% RSLogix 500 project MDM UPGRADE - onsite 5-11-08.RSS, saved by version 7.00.00.19 %
PROJECT "UNTITLED"    % processor: MicroLogix 1200 %

PROGRAM FILES
  LAD 2 "MAIN"  10 rungs
  LAD 3 "SEQUENCE"  61 rungs
  LAD 4 "OUTPUTS"  12 rungs

DATA FILES
  O0 OUTPUT  4 elements
  I1 INPUT  4 elements
  S2 STATUS  66 elements
  B3 BINARY  4 elements
  T4 TIMER  3 elements
  C5 COUNTER  1 elements
  R6 CONTROL  1 elements
  N7 INTEGER  7 elements
  F8 FLOAT  1 elements
  N9 SEQ TIMES  100 elements

LADDER 2 "MAIN"
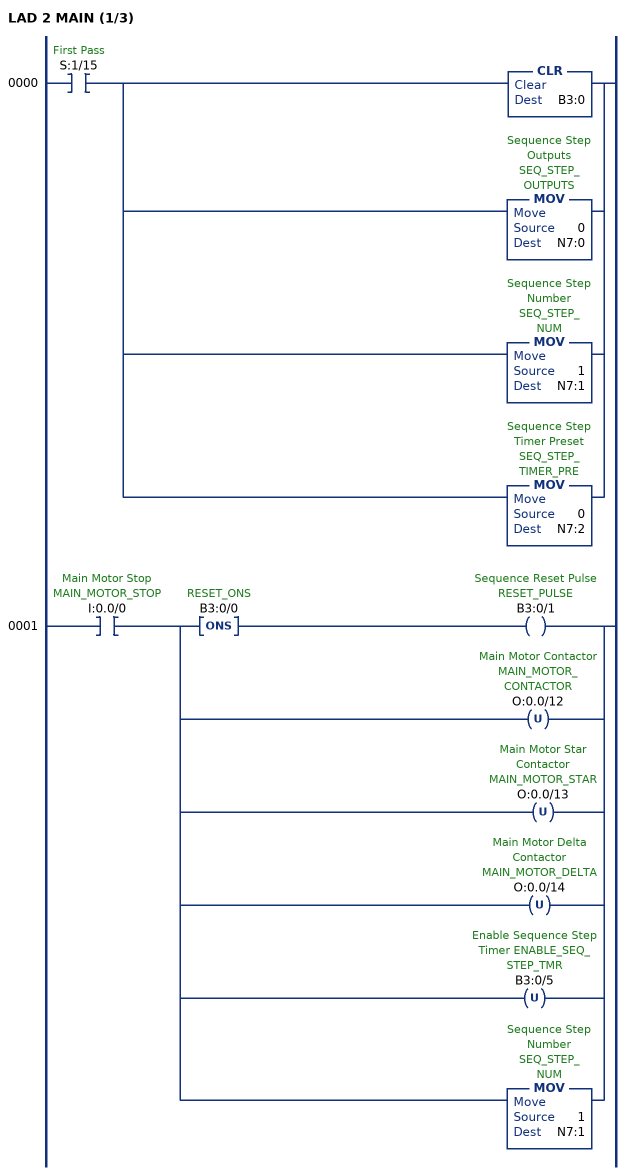
% Rung: 0 %
SOR XIC S:1/15 BST CLR B3:0 NXB MOV 0 N7:0 NXB MOV 1 N7:1 NXB MOV 0 N7:2 BND EOR
%   S:1/15  "First Pass" %
%   N7:0  SEQ_STEP_OUTPUTS  "Sequence Step Outputs" %
%   N7:1  SEQ_STEP_NUM  "Sequence Step Number" %
%   N7:2  SEQ_STEP_TIMER_PRE  "Sequence Step Timer Preset" %
% Rung: 1 %
SOR XIC I:0.0/0 BST ONS B3:0/0 OTE B3:0/1 NXB OTU O:0.0/12 NXB OTU O:0.0/13 NXB OTU O:0.0/14 NXB OTU B3:0/5 NXB MOV 1 N7:1 BND EOR
%   I:0.0/0  MAIN_MOTOR_STOP  "Main Motor Stop" %
%   B3:0/0  RESET_ONS %
%   B3:0/1  RESET_PULSE  "Sequence Reset Pulse" %
%   O:0.0/12  MAIN_MOTOR_CONTACTOR  "Main Motor Contactor" %
%   O:0.0/13  MAIN_MOTOR_STAR  "Main Motor Star Contactor" %
%   O:0.0/14  MAIN_MOTOR_DELTA  "Main Motor Delta Contactor" %
%   B3:0/5  ENABLE_SEQ_STEP_TMR  "Enable Sequence Step Timer" %
%   N7:1  SEQ_STEP_NUM  "Sequence Step Number" %

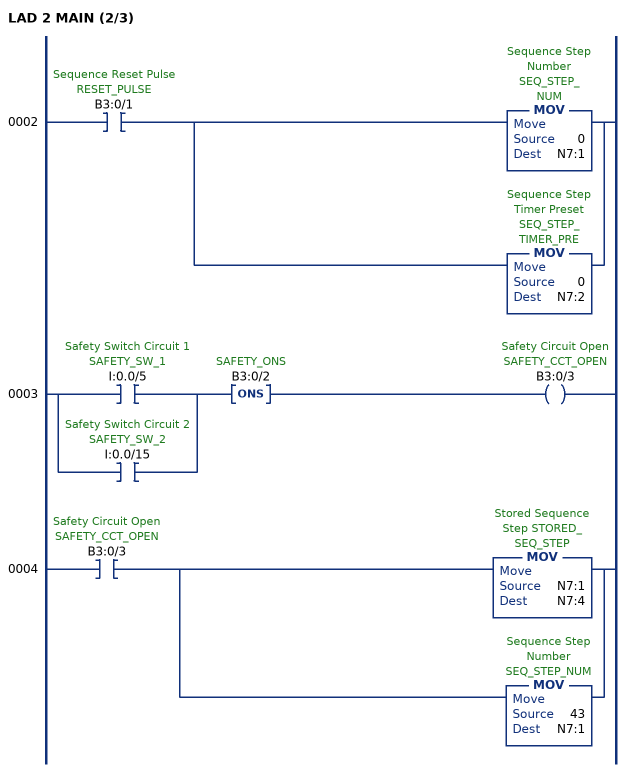
% Rung: 2 %
SOR XIC B3:0/1 BST MOV 0 N7:1 NXB MOV 0 N7:2 BND EOR
%   B3:0/1  RESET_PULSE  "Sequence Reset Pulse" %
%   N7:1  SEQ_STEP_NUM  "Sequence Step Number" %
%   N7:2  SEQ_STEP_TIMER_PRE  "Sequence Step Timer Preset" %
% Rung: 3 %
SOR BST XIC I:0.0/5 NXB XIC I:0.0/15 BND ONS B3:0/2 OTE B3:0/3 EOR
%   I:0.0/5  SAFETY_SW_1  "Safety Switch Circuit 1" %
%   I:0.0/15  SAFETY_SW_2  "Safety Switch Circuit 2" %
%   B3:0/2  SAFETY_ONS %
%   B3:0/3  SAFETY_CCT_OPEN  "Safety Circuit Open" %
% Rung: 4 %
SOR XIC B3:0/3 BST MOV N7:1 N7:4 NXB MOV 43 N7:1 BND EOR
%   B3:0/3  SAFETY_CCT_OPEN  "Safety Circuit Open" %
%   N7:1  SEQ_STEP_NUM  "Sequence Step Number" %
%   N7:4  STORED_SEQ_STEP  "Stored Sequence Step" %

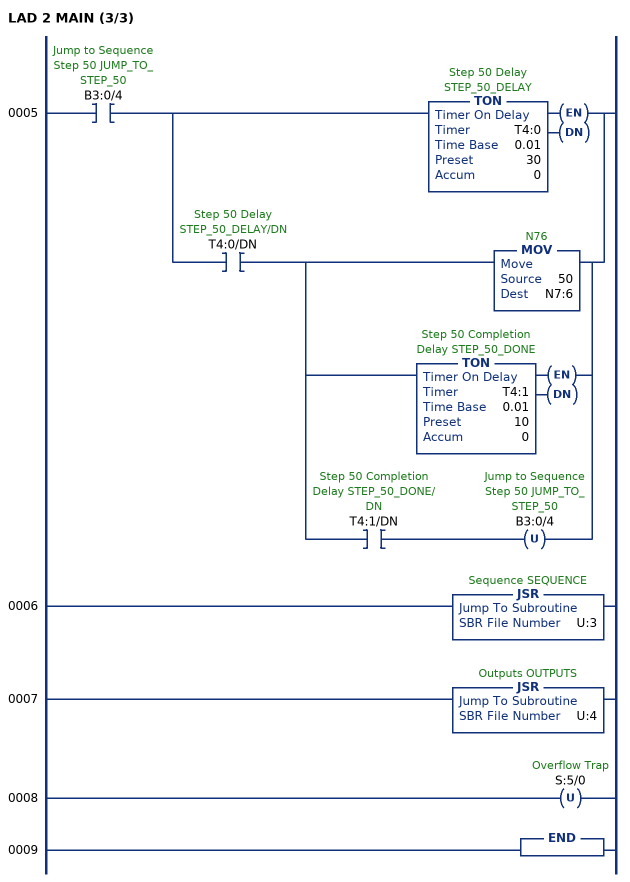
% Rung: 5 %
SOR XIC B3:0/4 BST TON T4:0 0.01 30 0 NXB XIC T4:0/DN BST MOV 50 N7:6 NXB TON T4:1 0.01 10 0 NXB XIC T4:1/DN OTU B3:0/4 BND BND EOR
%   B3:0/4  JUMP_TO_STEP_50  "Jump to Sequence Step 50" %
%   T4:0  STEP_50_DELAY  "Step 50 Delay" %
%   N7:6  N76 %
%   T4:1  STEP_50_DONE  "Step 50 Completion Delay" %
% Rung: 6 %
SOR JSR U:3 EOR
%   U:3  SEQUENCE  "Sequence" %
% Rung: 7 %
SOR JSR U:4 EOR
%   U:4  OUTPUTS  "Outputs" %
% Rung: 8 %
SOR OTU S:5/0 EOR
%   S:5/0  "Overflow Trap" %
% Rung: 9 %
SOR END EOR

LADDER 3 "SEQUENCE"
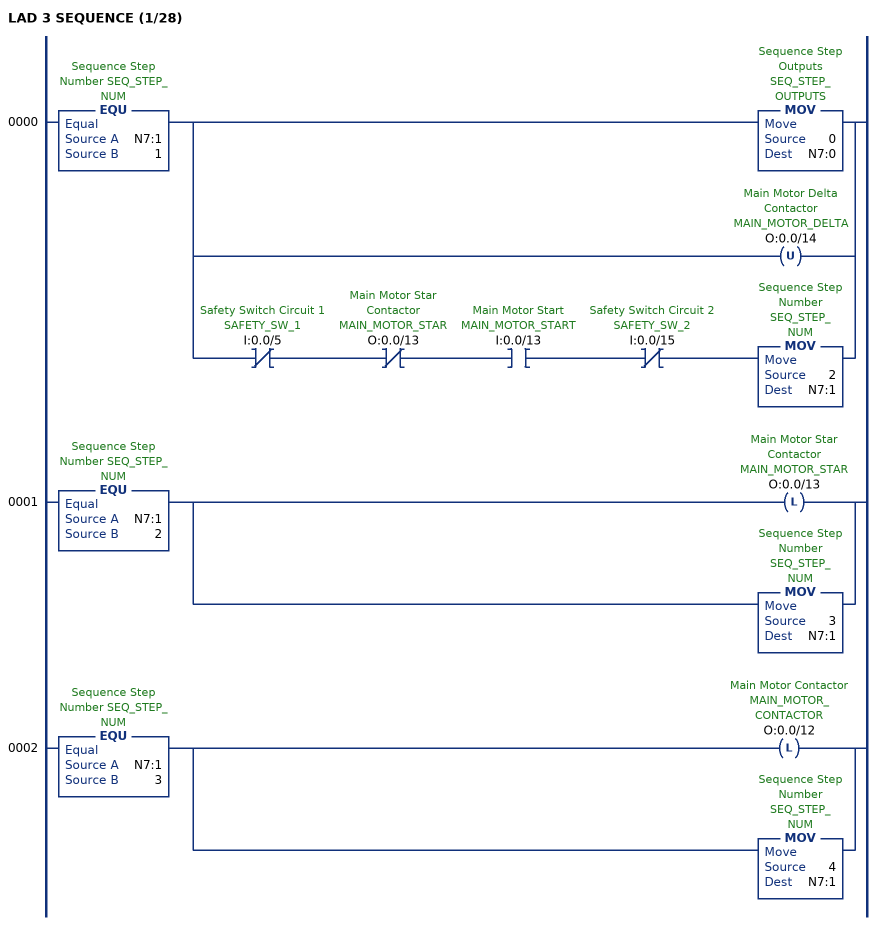
% Rung: 0 %
SOR EQU N7:1 1 BST MOV 0 N7:0 NXB OTU O:0.0/14 NXB XIO I:0.0/5 XIO O:0.0/13 XIC I:0.0/13 XIO I:0.0/15 MOV 2 N7:1 BND EOR
%   N7:1  SEQ_STEP_NUM  "Sequence Step Number" %
%   N7:0  SEQ_STEP_OUTPUTS  "Sequence Step Outputs" %
%   O:0.0/14  MAIN_MOTOR_DELTA  "Main Motor Delta Contactor" %
%   I:0.0/5  SAFETY_SW_1  "Safety Switch Circuit 1" %
%   O:0.0/13  MAIN_MOTOR_STAR  "Main Motor Star Contactor" %
%   I:0.0/13  MAIN_MOTOR_START  "Main Motor Start" %
%   I:0.0/15  SAFETY_SW_2  "Safety Switch Circuit 2" %
% Rung: 1 %
SOR EQU N7:1 2 BST OTL O:0.0/13 NXB MOV 3 N7:1 BND EOR
%   N7:1  SEQ_STEP_NUM  "Sequence Step Number" %
%   O:0.0/13  MAIN_MOTOR_STAR  "Main Motor Star Contactor" %
% Rung: 2 %
SOR EQU N7:1 3 BST OTL O:0.0/12 NXB MOV 4 N7:1 BND EOR
%   N7:1  SEQ_STEP_NUM  "Sequence Step Number" %
%   O:0.0/12  MAIN_MOTOR_CONTACTOR  "Main Motor Contactor" %

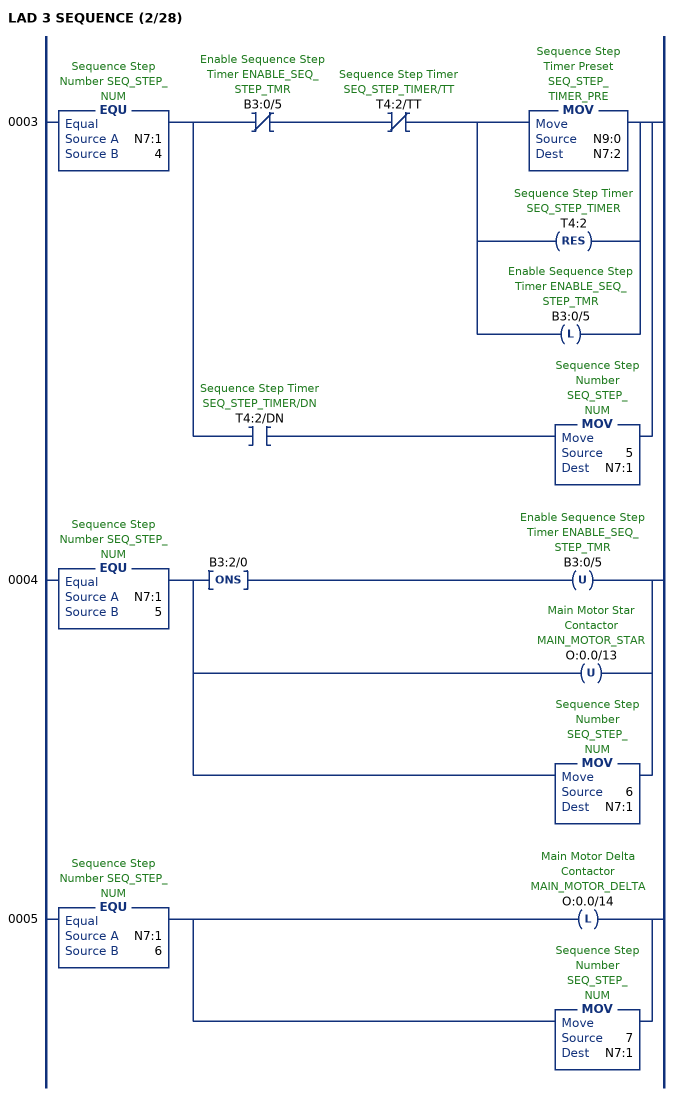
% Rung: 3 %
SOR EQU N7:1 4 BST XIO B3:0/5 XIO T4:2/TT BST MOV N9:0 N7:2 NXB RES T4:2 NXB OTL B3:0/5 BND NXB XIC T4:2/DN MOV 5 N7:1 BND EOR
%   N7:1  SEQ_STEP_NUM  "Sequence Step Number" %
%   B3:0/5  ENABLE_SEQ_STEP_TMR  "Enable Sequence Step Timer" %
%   T4:2  SEQ_STEP_TIMER  "Sequence Step Timer" %
%   N7:2  SEQ_STEP_TIMER_PRE  "Sequence Step Timer Preset" %
% Rung: 4 %
SOR EQU N7:1 5 BST ONS B3:2/0 OTU B3:0/5 NXB OTU O:0.0/13 NXB MOV 6 N7:1 BND EOR
%   N7:1  SEQ_STEP_NUM  "Sequence Step Number" %
%   B3:0/5  ENABLE_SEQ_STEP_TMR  "Enable Sequence Step Timer" %
%   O:0.0/13  MAIN_MOTOR_STAR  "Main Motor Star Contactor" %
% Rung: 5 %
SOR EQU N7:1 6 BST OTL O:0.0/14 NXB MOV 7 N7:1 BND EOR
%   N7:1  SEQ_STEP_NUM  "Sequence Step Number" %
%   O:0.0/14  MAIN_MOTOR_DELTA  "Main Motor Delta Contactor" %

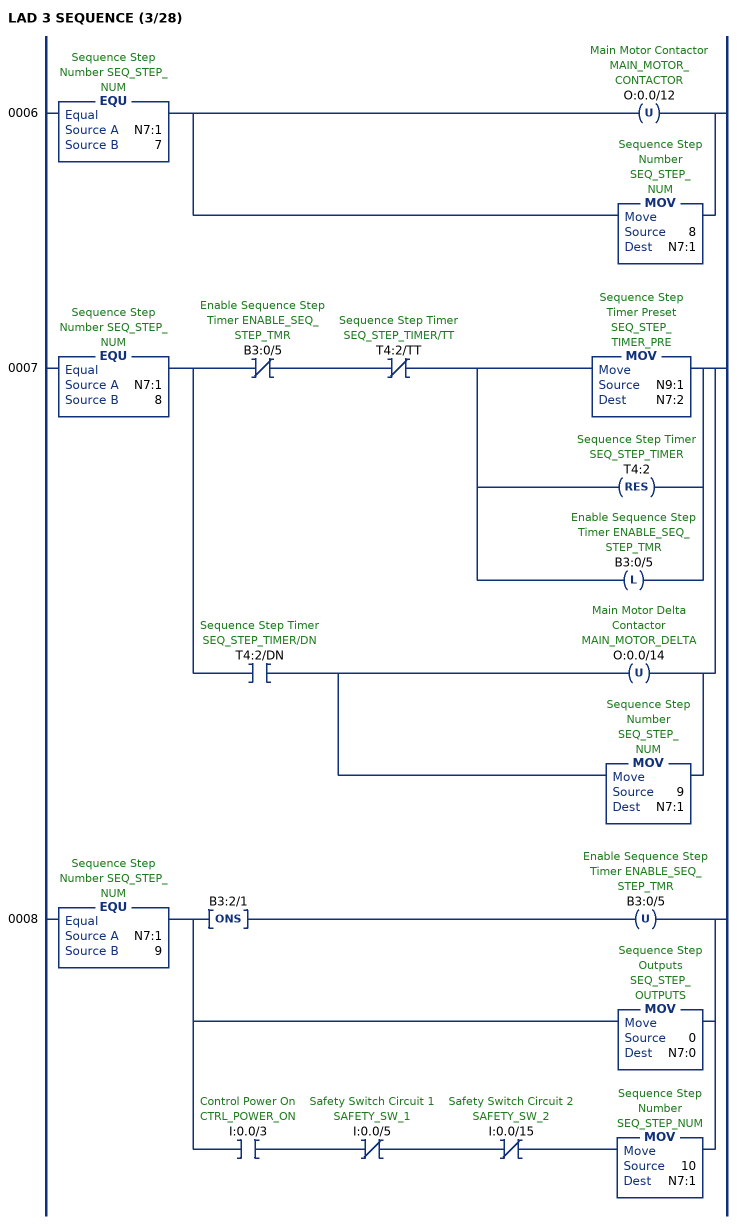
% Rung: 6 %
SOR EQU N7:1 7 BST OTU O:0.0/12 NXB MOV 8 N7:1 BND EOR
%   N7:1  SEQ_STEP_NUM  "Sequence Step Number" %
%   O:0.0/12  MAIN_MOTOR_CONTACTOR  "Main Motor Contactor" %
% Rung: 7 %
SOR EQU N7:1 8 BST XIO B3:0/5 XIO T4:2/TT BST MOV N9:1 N7:2 NXB RES T4:2 NXB OTL B3:0/5 BND NXB XIC T4:2/DN BST OTU O:0.0/14 NXB MOV 9 N7:1 BND BND EOR
%   N7:1  SEQ_STEP_NUM  "Sequence Step Number" %
%   B3:0/5  ENABLE_SEQ_STEP_TMR  "Enable Sequence Step Timer" %
%   T4:2  SEQ_STEP_TIMER  "Sequence Step Timer" %
%   N7:2  SEQ_STEP_TIMER_PRE  "Sequence Step Timer Preset" %
%   O:0.0/14  MAIN_MOTOR_DELTA  "Main Motor Delta Contactor" %
% Rung: 8 %
SOR EQU N7:1 9 BST ONS B3:2/1 OTU B3:0/5 NXB MOV 0 N7:0 NXB XIC I:0.0/3 XIO I:0.0/5 XIO I:0.0/15 MOV 10 N7:1 BND EOR
%   N7:1  SEQ_STEP_NUM  "Sequence Step Number" %
%   B3:0/5  ENABLE_SEQ_STEP_TMR  "Enable Sequence Step Timer" %
%   N7:0  SEQ_STEP_OUTPUTS  "Sequence Step Outputs" %
%   I:0.0/3  CTRL_POWER_ON  "Control Power On" %
%   I:0.0/5  SAFETY_SW_1  "Safety Switch Circuit 1" %
%   I:0.0/15  SAFETY_SW_2  "Safety Switch Circuit 2" %

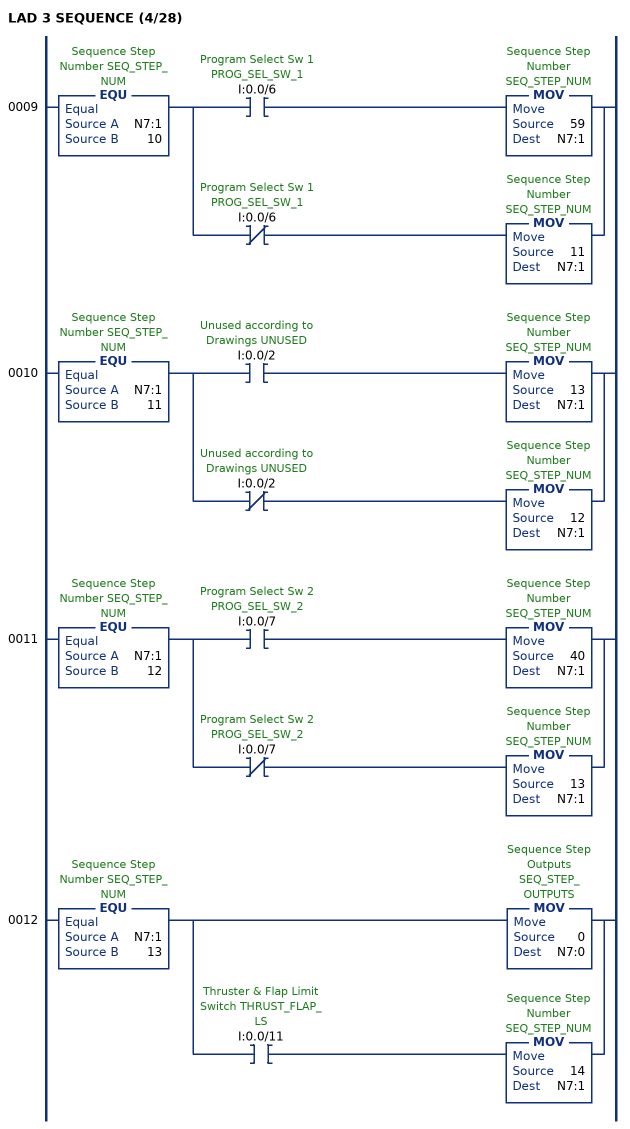
% Rung: 9 %
SOR EQU N7:1 10 BST XIC I:0.0/6 MOV 59 N7:1 NXB XIO I:0.0/6 MOV 11 N7:1 BND EOR
%   N7:1  SEQ_STEP_NUM  "Sequence Step Number" %
%   I:0.0/6  PROG_SEL_SW_1  "Program Select Sw 1" %
% Rung: 10 %
SOR EQU N7:1 11 BST XIC I:0.0/2 MOV 13 N7:1 NXB XIO I:0.0/2 MOV 12 N7:1 BND EOR
%   N7:1  SEQ_STEP_NUM  "Sequence Step Number" %
%   I:0.0/2  UNUSED  "Unused according to Drawings" %
% Rung: 11 %
SOR EQU N7:1 12 BST XIC I:0.0/7 MOV 40 N7:1 NXB XIO I:0.0/7 MOV 13 N7:1 BND EOR
%   N7:1  SEQ_STEP_NUM  "Sequence Step Number" %
%   I:0.0/7  PROG_SEL_SW_2  "Program Select Sw 2" %
% Rung: 12 %
SOR EQU N7:1 13 BST MOV 0 N7:0 NXB XIC I:0.0/11 MOV 14 N7:1 BND EOR
%   N7:1  SEQ_STEP_NUM  "Sequence Step Number" %
%   N7:0  SEQ_STEP_OUTPUTS  "Sequence Step Outputs" %
%   I:0.0/11  THRUST_FLAP_LS  "Thruster & Flap Limit Switch" %

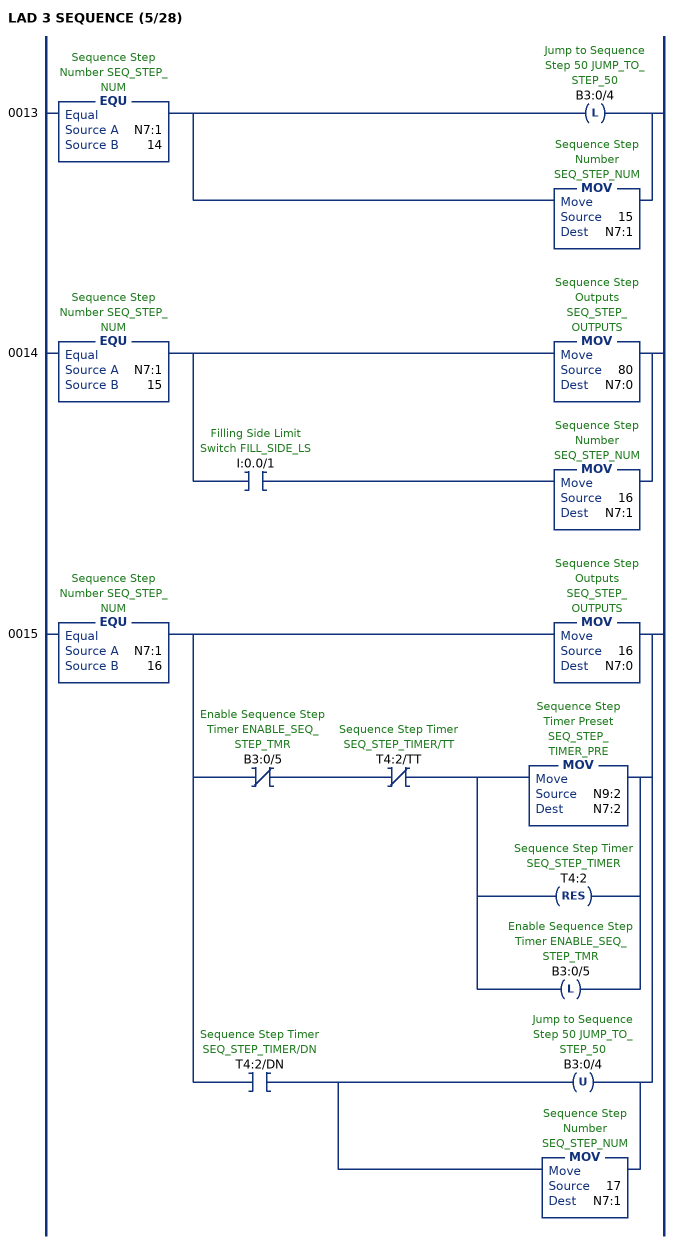
% Rung: 13 %
SOR EQU N7:1 14 BST OTL B3:0/4 NXB MOV 15 N7:1 BND EOR
%   N7:1  SEQ_STEP_NUM  "Sequence Step Number" %
%   B3:0/4  JUMP_TO_STEP_50  "Jump to Sequence Step 50" %
% Rung: 14 %
SOR EQU N7:1 15 BST MOV 80 N7:0 NXB XIC I:0.0/1 MOV 16 N7:1 BND EOR
%   N7:1  SEQ_STEP_NUM  "Sequence Step Number" %
%   N7:0  SEQ_STEP_OUTPUTS  "Sequence Step Outputs" %
%   I:0.0/1  FILL_SIDE_LS  "Filling Side Limit Switch" %
% Rung: 15 %
SOR EQU N7:1 16 BST MOV 16 N7:0 NXB XIO B3:0/5 XIO T4:2/TT BST MOV N9:2 N7:2 NXB RES T4:2 NXB OTL B3:0/5 BND NXB XIC T4:2/DN BST OTU B3:0/4 NXB MOV 17 N7:1 BND BND EOR
%   N7:1  SEQ_STEP_NUM  "Sequence Step Number" %
%   N7:0  SEQ_STEP_OUTPUTS  "Sequence Step Outputs" %
%   B3:0/5  ENABLE_SEQ_STEP_TMR  "Enable Sequence Step Timer" %
%   T4:2  SEQ_STEP_TIMER  "Sequence Step Timer" %
%   N7:2  SEQ_STEP_TIMER_PRE  "Sequence Step Timer Preset" %
%   B3:0/4  JUMP_TO_STEP_50  "Jump to Sequence Step 50" %

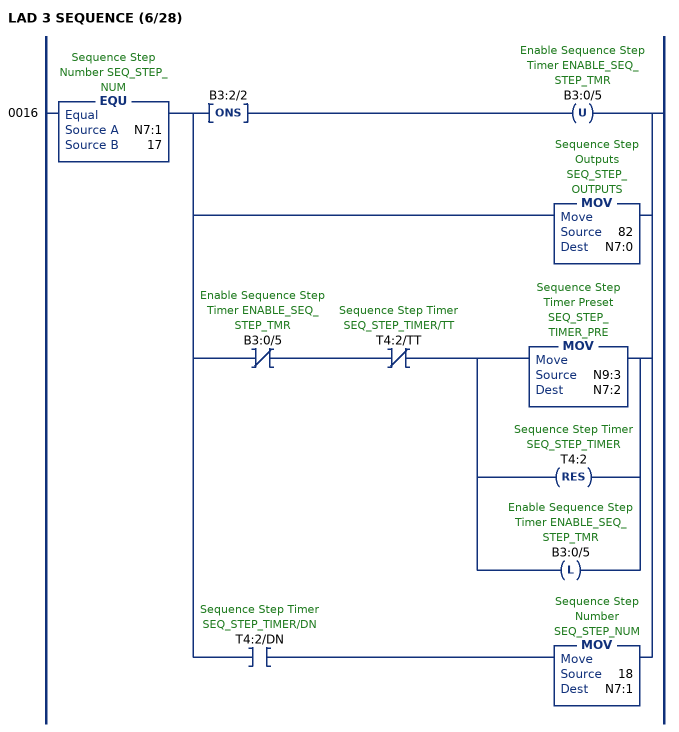
% Rung: 16 %
SOR EQU N7:1 17 BST ONS B3:2/2 OTU B3:0/5 NXB MOV 82 N7:0 NXB XIO B3:0/5 XIO T4:2/TT BST MOV N9:3 N7:2 NXB RES T4:2 NXB OTL B3:0/5 BND NXB XIC T4:2/DN MOV 18 N7:1 BND EOR
%   N7:1  SEQ_STEP_NUM  "Sequence Step Number" %
%   B3:0/5  ENABLE_SEQ_STEP_TMR  "Enable Sequence Step Timer" %
%   N7:0  SEQ_STEP_OUTPUTS  "Sequence Step Outputs" %
%   T4:2  SEQ_STEP_TIMER  "Sequence Step Timer" %
%   N7:2  SEQ_STEP_TIMER_PRE  "Sequence Step Timer Preset" %

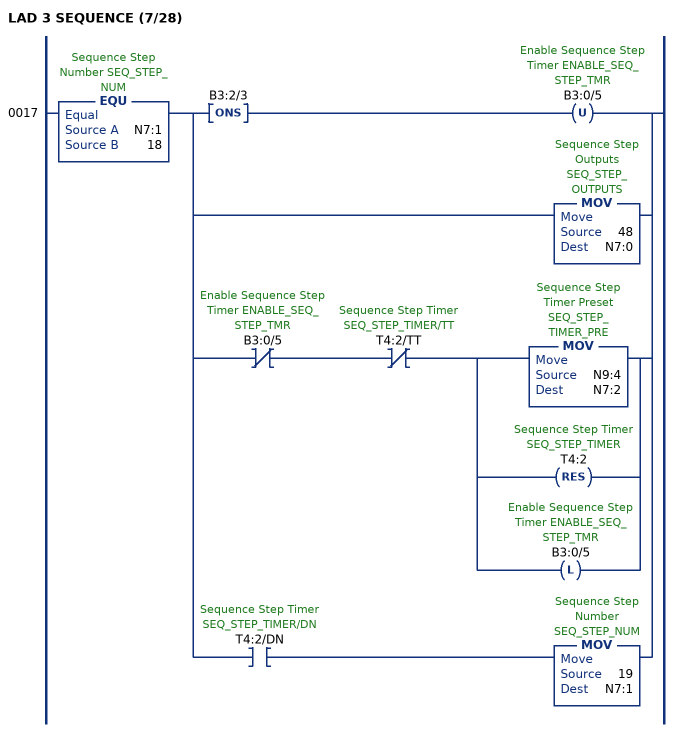
% Rung: 17 %
SOR EQU N7:1 18 BST ONS B3:2/3 OTU B3:0/5 NXB MOV 48 N7:0 NXB XIO B3:0/5 XIO T4:2/TT BST MOV N9:4 N7:2 NXB RES T4:2 NXB OTL B3:0/5 BND NXB XIC T4:2/DN MOV 19 N7:1 BND EOR
%   N7:1  SEQ_STEP_NUM  "Sequence Step Number" %
%   B3:0/5  ENABLE_SEQ_STEP_TMR  "Enable Sequence Step Timer" %
%   N7:0  SEQ_STEP_OUTPUTS  "Sequence Step Outputs" %
%   T4:2  SEQ_STEP_TIMER  "Sequence Step Timer" %
%   N7:2  SEQ_STEP_TIMER_PRE  "Sequence Step Timer Preset" %

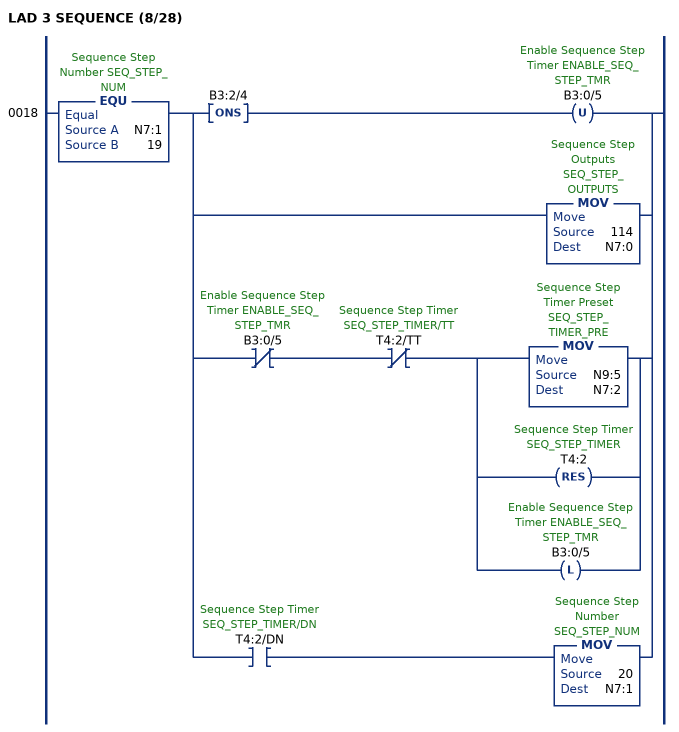
% Rung: 18 %
SOR EQU N7:1 19 BST ONS B3:2/4 OTU B3:0/5 NXB MOV 114 N7:0 NXB XIO B3:0/5 XIO T4:2/TT BST MOV N9:5 N7:2 NXB RES T4:2 NXB OTL B3:0/5 BND NXB XIC T4:2/DN MOV 20 N7:1 BND EOR
%   N7:1  SEQ_STEP_NUM  "Sequence Step Number" %
%   B3:0/5  ENABLE_SEQ_STEP_TMR  "Enable Sequence Step Timer" %
%   N7:0  SEQ_STEP_OUTPUTS  "Sequence Step Outputs" %
%   T4:2  SEQ_STEP_TIMER  "Sequence Step Timer" %
%   N7:2  SEQ_STEP_TIMER_PRE  "Sequence Step Timer Preset" %

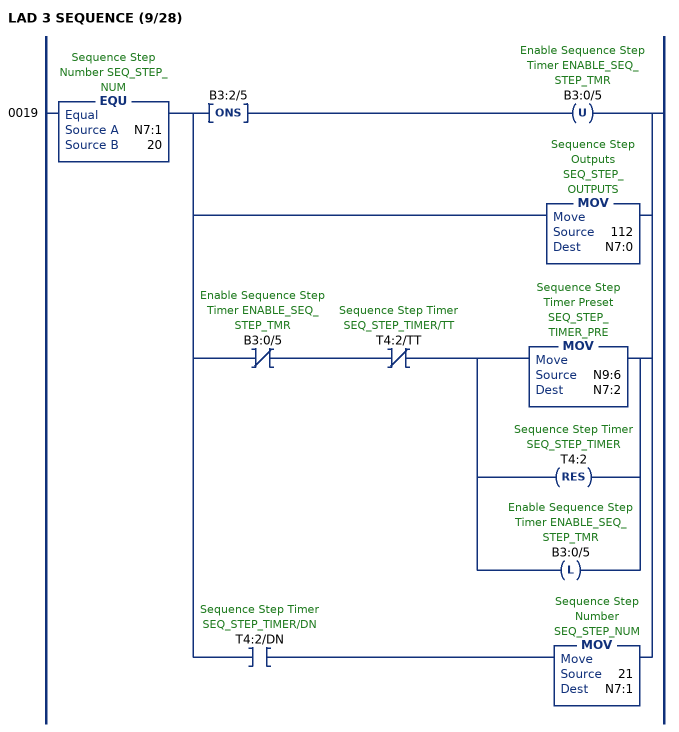
% Rung: 19 %
SOR EQU N7:1 20 BST ONS B3:2/5 OTU B3:0/5 NXB MOV 112 N7:0 NXB XIO B3:0/5 XIO T4:2/TT BST MOV N9:6 N7:2 NXB RES T4:2 NXB OTL B3:0/5 BND NXB XIC T4:2/DN MOV 21 N7:1 BND EOR
%   N7:1  SEQ_STEP_NUM  "Sequence Step Number" %
%   B3:0/5  ENABLE_SEQ_STEP_TMR  "Enable Sequence Step Timer" %
%   N7:0  SEQ_STEP_OUTPUTS  "Sequence Step Outputs" %
%   T4:2  SEQ_STEP_TIMER  "Sequence Step Timer" %
%   N7:2  SEQ_STEP_TIMER_PRE  "Sequence Step Timer Preset" %

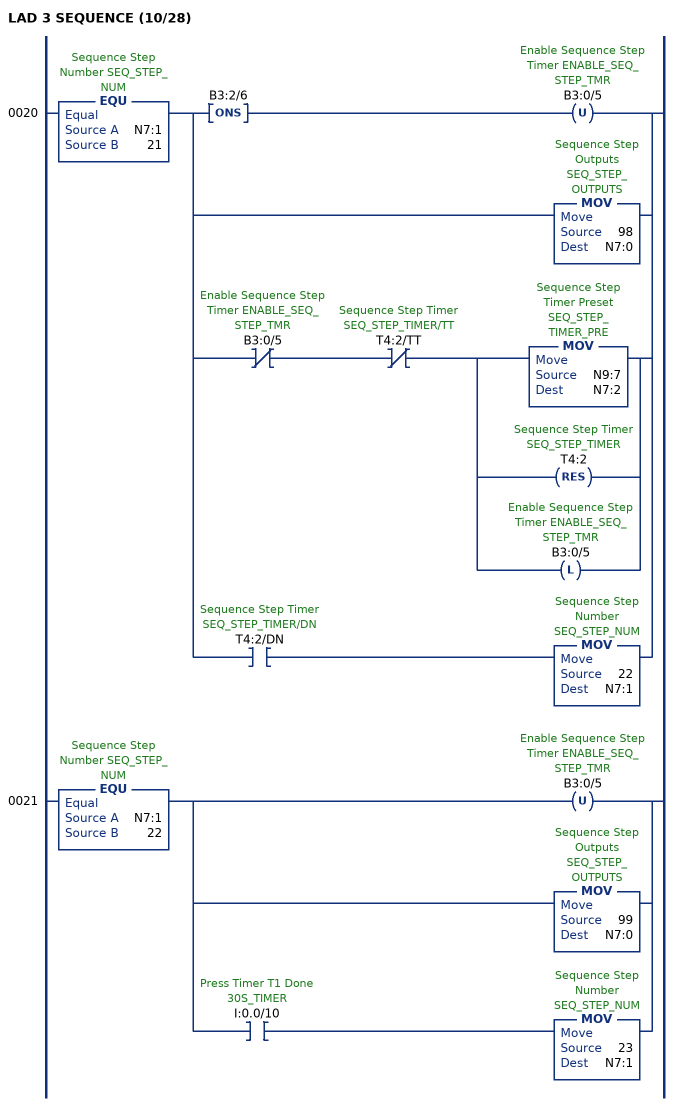
% Rung: 20 %
SOR EQU N7:1 21 BST ONS B3:2/6 OTU B3:0/5 NXB MOV 98 N7:0 NXB XIO B3:0/5 XIO T4:2/TT BST MOV N9:7 N7:2 NXB RES T4:2 NXB OTL B3:0/5 BND NXB XIC T4:2/DN MOV 22 N7:1 BND EOR
%   N7:1  SEQ_STEP_NUM  "Sequence Step Number" %
%   B3:0/5  ENABLE_SEQ_STEP_TMR  "Enable Sequence Step Timer" %
%   N7:0  SEQ_STEP_OUTPUTS  "Sequence Step Outputs" %
%   T4:2  SEQ_STEP_TIMER  "Sequence Step Timer" %
%   N7:2  SEQ_STEP_TIMER_PRE  "Sequence Step Timer Preset" %
% Rung: 21 %
SOR EQU N7:1 22 BST OTU B3:0/5 NXB MOV 99 N7:0 NXB XIC I:0.0/10 MOV 23 N7:1 BND EOR
%   N7:1  SEQ_STEP_NUM  "Sequence Step Number" %
%   B3:0/5  ENABLE_SEQ_STEP_TMR  "Enable Sequence Step Timer" %
%   N7:0  SEQ_STEP_OUTPUTS  "Sequence Step Outputs" %
%   I:0.0/10  30S_TIMER  "Press Timer T1 Done" %

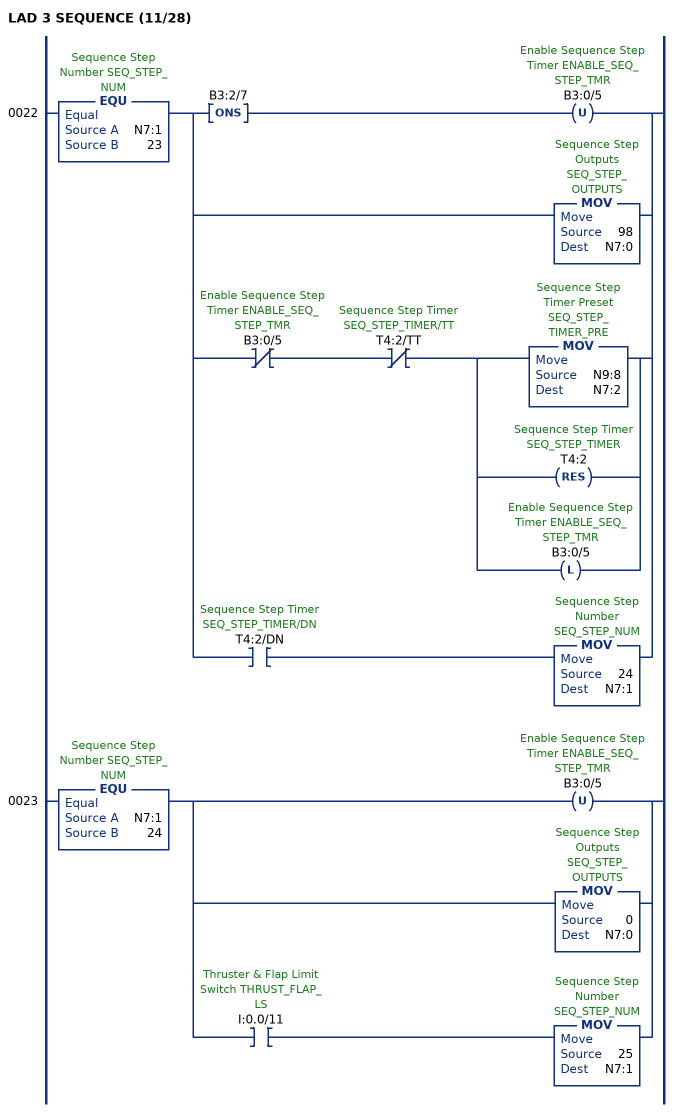
% Rung: 22 %
SOR EQU N7:1 23 BST ONS B3:2/7 OTU B3:0/5 NXB MOV 98 N7:0 NXB XIO B3:0/5 XIO T4:2/TT BST MOV N9:8 N7:2 NXB RES T4:2 NXB OTL B3:0/5 BND NXB XIC T4:2/DN MOV 24 N7:1 BND EOR
%   N7:1  SEQ_STEP_NUM  "Sequence Step Number" %
%   B3:0/5  ENABLE_SEQ_STEP_TMR  "Enable Sequence Step Timer" %
%   N7:0  SEQ_STEP_OUTPUTS  "Sequence Step Outputs" %
%   T4:2  SEQ_STEP_TIMER  "Sequence Step Timer" %
%   N7:2  SEQ_STEP_TIMER_PRE  "Sequence Step Timer Preset" %
% Rung: 23 %
SOR EQU N7:1 24 BST OTU B3:0/5 NXB MOV 0 N7:0 NXB XIC I:0.0/11 MOV 25 N7:1 BND EOR
%   N7:1  SEQ_STEP_NUM  "Sequence Step Number" %
%   B3:0/5  ENABLE_SEQ_STEP_TMR  "Enable Sequence Step Timer" %
%   N7:0  SEQ_STEP_OUTPUTS  "Sequence Step Outputs" %
%   I:0.0/11  THRUST_FLAP_LS  "Thruster & Flap Limit Switch" %

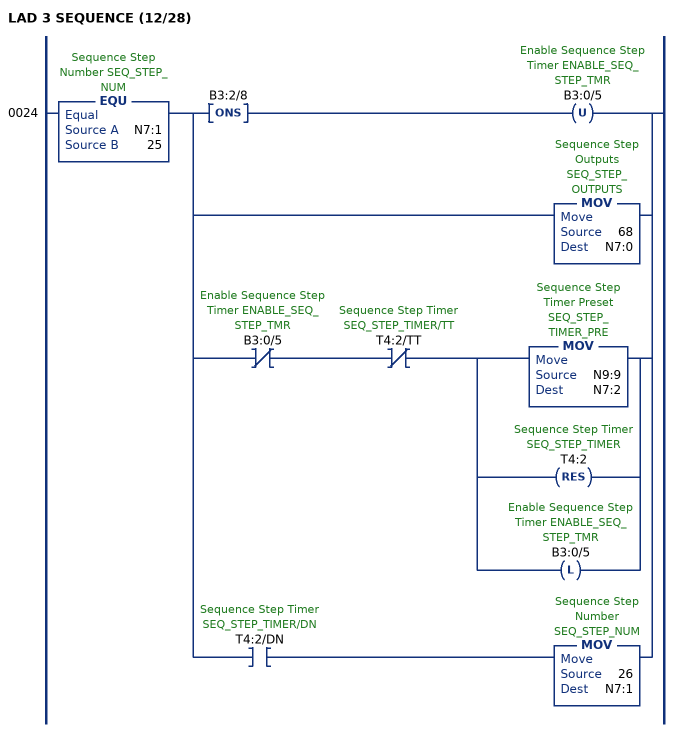
% Rung: 24 %
SOR EQU N7:1 25 BST ONS B3:2/8 OTU B3:0/5 NXB MOV 68 N7:0 NXB XIO B3:0/5 XIO T4:2/TT BST MOV N9:9 N7:2 NXB RES T4:2 NXB OTL B3:0/5 BND NXB XIC T4:2/DN MOV 26 N7:1 BND EOR
%   N7:1  SEQ_STEP_NUM  "Sequence Step Number" %
%   B3:0/5  ENABLE_SEQ_STEP_TMR  "Enable Sequence Step Timer" %
%   N7:0  SEQ_STEP_OUTPUTS  "Sequence Step Outputs" %
%   T4:2  SEQ_STEP_TIMER  "Sequence Step Timer" %
%   N7:2  SEQ_STEP_TIMER_PRE  "Sequence Step Timer Preset" %

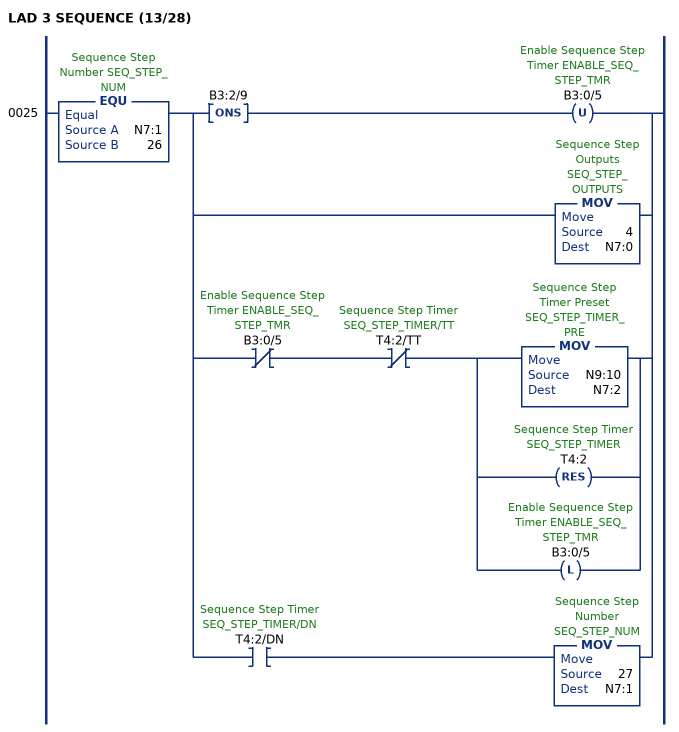
% Rung: 25 %
SOR EQU N7:1 26 BST ONS B3:2/9 OTU B3:0/5 NXB MOV 4 N7:0 NXB XIO B3:0/5 XIO T4:2/TT BST MOV N9:10 N7:2 NXB RES T4:2 NXB OTL B3:0/5 BND NXB XIC T4:2/DN MOV 27 N7:1 BND EOR
%   N7:1  SEQ_STEP_NUM  "Sequence Step Number" %
%   B3:0/5  ENABLE_SEQ_STEP_TMR  "Enable Sequence Step Timer" %
%   N7:0  SEQ_STEP_OUTPUTS  "Sequence Step Outputs" %
%   T4:2  SEQ_STEP_TIMER  "Sequence Step Timer" %
%   N7:2  SEQ_STEP_TIMER_PRE  "Sequence Step Timer Preset" %

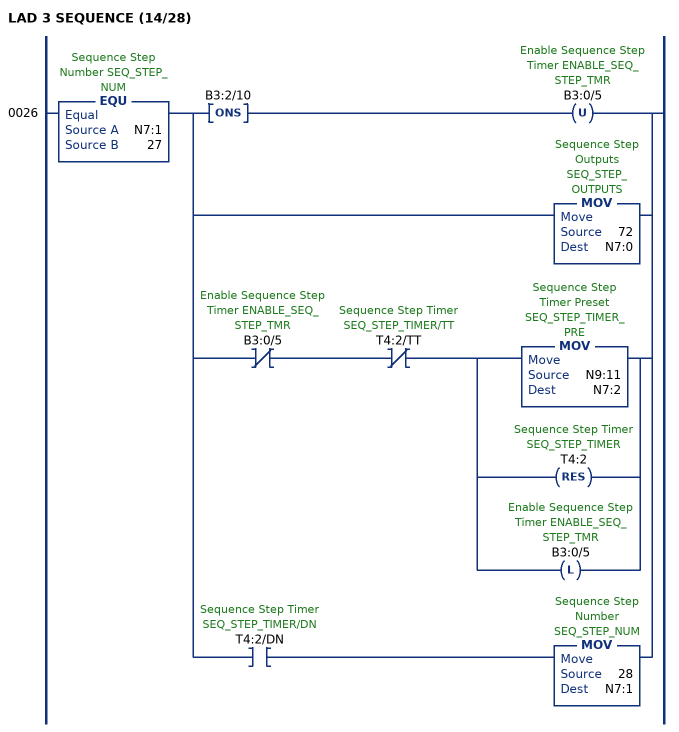
% Rung: 26 %
SOR EQU N7:1 27 BST ONS B3:2/10 OTU B3:0/5 NXB MOV 72 N7:0 NXB XIO B3:0/5 XIO T4:2/TT BST MOV N9:11 N7:2 NXB RES T4:2 NXB OTL B3:0/5 BND NXB XIC T4:2/DN MOV 28 N7:1 BND EOR
%   N7:1  SEQ_STEP_NUM  "Sequence Step Number" %
%   B3:0/5  ENABLE_SEQ_STEP_TMR  "Enable Sequence Step Timer" %
%   N7:0  SEQ_STEP_OUTPUTS  "Sequence Step Outputs" %
%   T4:2  SEQ_STEP_TIMER  "Sequence Step Timer" %
%   N7:2  SEQ_STEP_TIMER_PRE  "Sequence Step Timer Preset" %

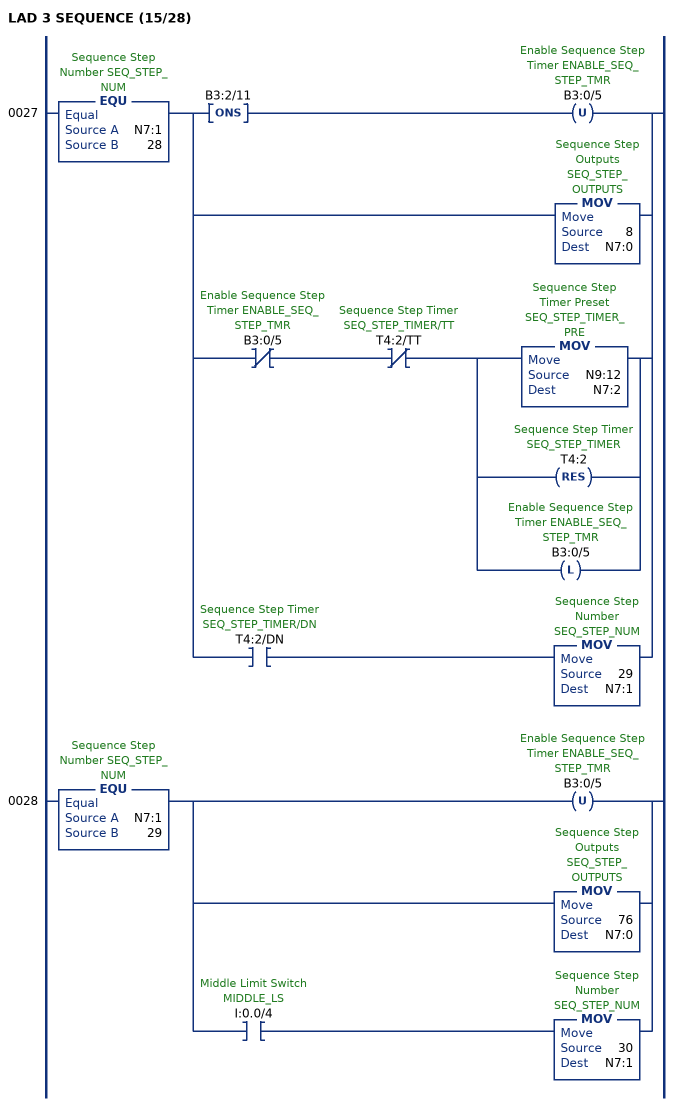
% Rung: 27 %
SOR EQU N7:1 28 BST ONS B3:2/11 OTU B3:0/5 NXB MOV 8 N7:0 NXB XIO B3:0/5 XIO T4:2/TT BST MOV N9:12 N7:2 NXB RES T4:2 NXB OTL B3:0/5 BND NXB XIC T4:2/DN MOV 29 N7:1 BND EOR
%   N7:1  SEQ_STEP_NUM  "Sequence Step Number" %
%   B3:0/5  ENABLE_SEQ_STEP_TMR  "Enable Sequence Step Timer" %
%   N7:0  SEQ_STEP_OUTPUTS  "Sequence Step Outputs" %
%   T4:2  SEQ_STEP_TIMER  "Sequence Step Timer" %
%   N7:2  SEQ_STEP_TIMER_PRE  "Sequence Step Timer Preset" %
% Rung: 28 %
SOR EQU N7:1 29 BST OTU B3:0/5 NXB MOV 76 N7:0 NXB XIC I:0.0/4 MOV 30 N7:1 BND EOR
%   N7:1  SEQ_STEP_NUM  "Sequence Step Number" %
%   B3:0/5  ENABLE_SEQ_STEP_TMR  "Enable Sequence Step Timer" %
%   N7:0  SEQ_STEP_OUTPUTS  "Sequence Step Outputs" %
%   I:0.0/4  MIDDLE_LS  "Middle Limit Switch" %

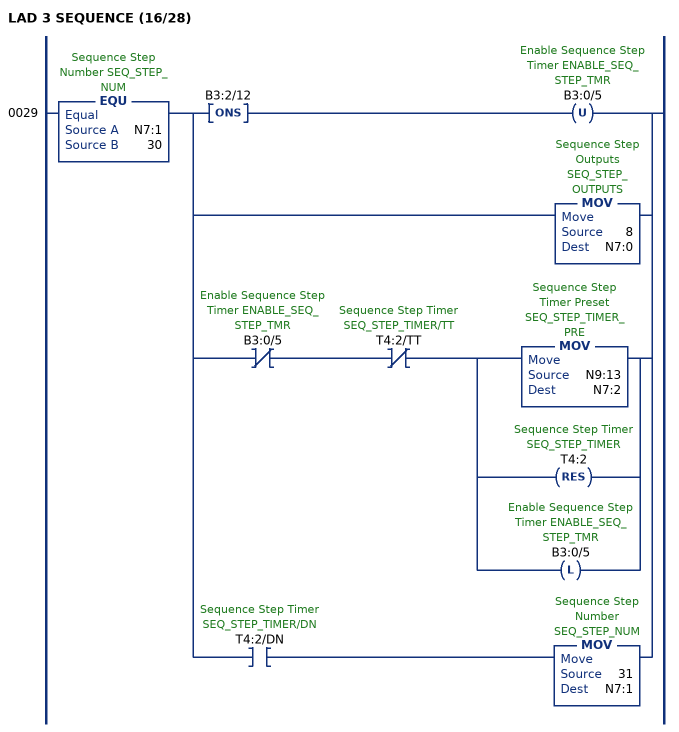
% Rung: 29 %
SOR EQU N7:1 30 BST ONS B3:2/12 OTU B3:0/5 NXB MOV 8 N7:0 NXB XIO B3:0/5 XIO T4:2/TT BST MOV N9:13 N7:2 NXB RES T4:2 NXB OTL B3:0/5 BND NXB XIC T4:2/DN MOV 31 N7:1 BND EOR
%   N7:1  SEQ_STEP_NUM  "Sequence Step Number" %
%   B3:0/5  ENABLE_SEQ_STEP_TMR  "Enable Sequence Step Timer" %
%   N7:0  SEQ_STEP_OUTPUTS  "Sequence Step Outputs" %
%   T4:2  SEQ_STEP_TIMER  "Sequence Step Timer" %
%   N7:2  SEQ_STEP_TIMER_PRE  "Sequence Step Timer Preset" %

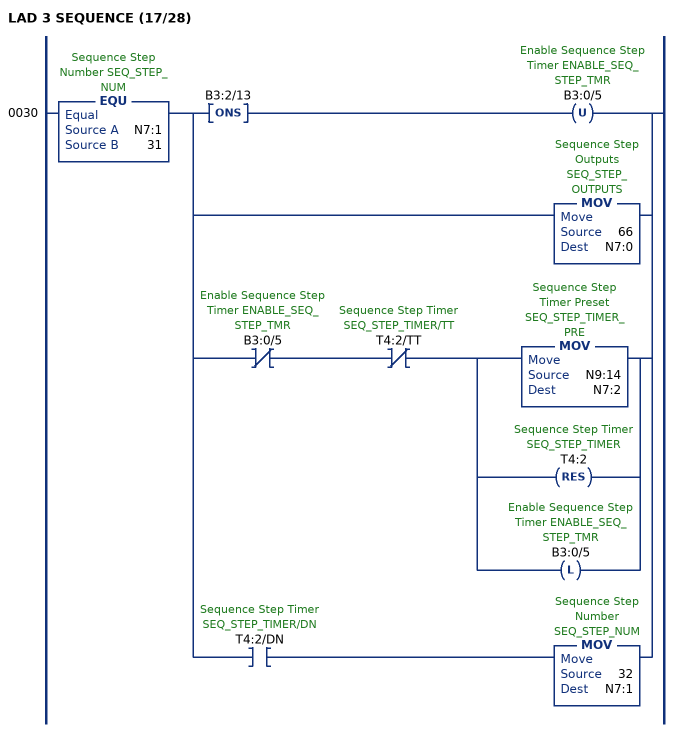
% Rung: 30 %
SOR EQU N7:1 31 BST ONS B3:2/13 OTU B3:0/5 NXB MOV 66 N7:0 NXB XIO B3:0/5 XIO T4:2/TT BST MOV N9:14 N7:2 NXB RES T4:2 NXB OTL B3:0/5 BND NXB XIC T4:2/DN MOV 32 N7:1 BND EOR
%   N7:1  SEQ_STEP_NUM  "Sequence Step Number" %
%   B3:0/5  ENABLE_SEQ_STEP_TMR  "Enable Sequence Step Timer" %
%   N7:0  SEQ_STEP_OUTPUTS  "Sequence Step Outputs" %
%   T4:2  SEQ_STEP_TIMER  "Sequence Step Timer" %
%   N7:2  SEQ_STEP_TIMER_PRE  "Sequence Step Timer Preset" %

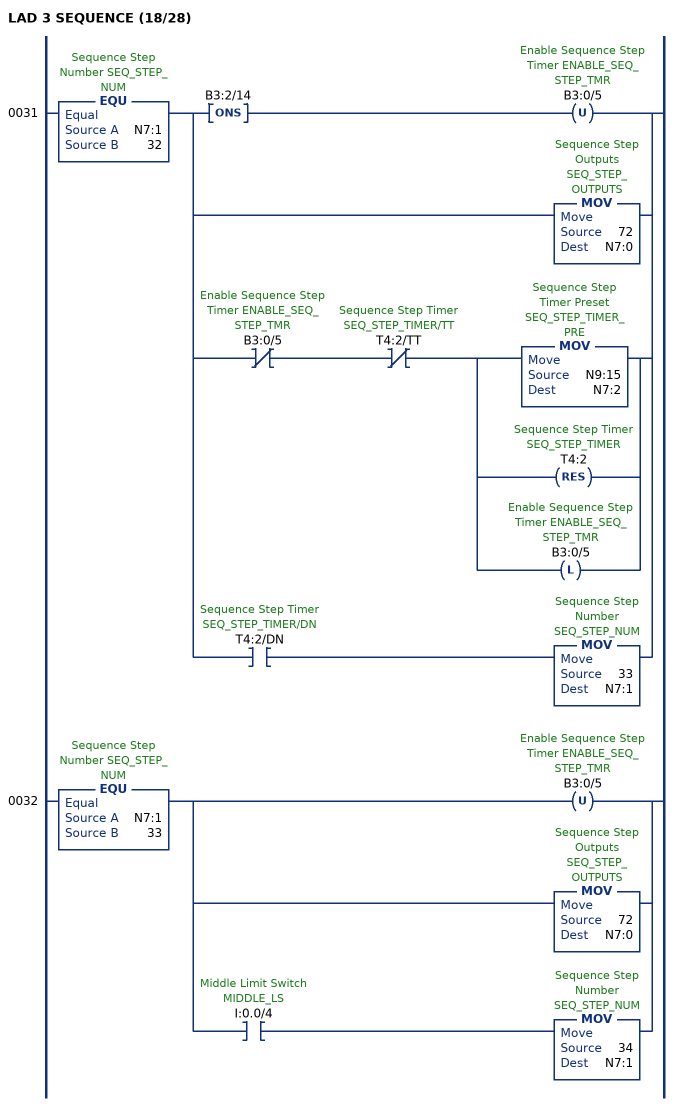
% Rung: 31 %
SOR EQU N7:1 32 BST ONS B3:2/14 OTU B3:0/5 NXB MOV 72 N7:0 NXB XIO B3:0/5 XIO T4:2/TT BST MOV N9:15 N7:2 NXB RES T4:2 NXB OTL B3:0/5 BND NXB XIC T4:2/DN MOV 33 N7:1 BND EOR
%   N7:1  SEQ_STEP_NUM  "Sequence Step Number" %
%   B3:0/5  ENABLE_SEQ_STEP_TMR  "Enable Sequence Step Timer" %
%   N7:0  SEQ_STEP_OUTPUTS  "Sequence Step Outputs" %
%   T4:2  SEQ_STEP_TIMER  "Sequence Step Timer" %
%   N7:2  SEQ_STEP_TIMER_PRE  "Sequence Step Timer Preset" %
% Rung: 32 %
SOR EQU N7:1 33 BST OTU B3:0/5 NXB MOV 72 N7:0 NXB XIC I:0.0/4 MOV 34 N7:1 BND EOR
%   N7:1  SEQ_STEP_NUM  "Sequence Step Number" %
%   B3:0/5  ENABLE_SEQ_STEP_TMR  "Enable Sequence Step Timer" %
%   N7:0  SEQ_STEP_OUTPUTS  "Sequence Step Outputs" %
%   I:0.0/4  MIDDLE_LS  "Middle Limit Switch" %

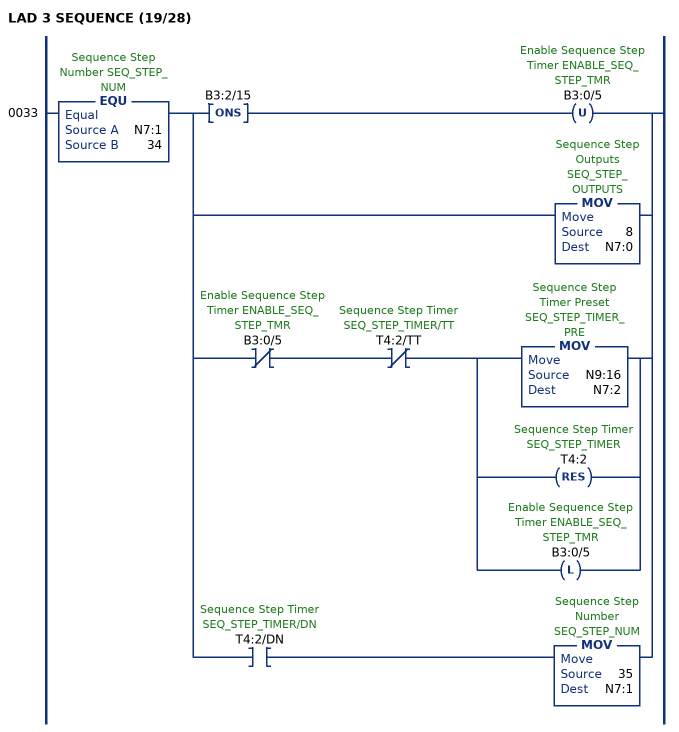
% Rung: 33 %
SOR EQU N7:1 34 BST ONS B3:2/15 OTU B3:0/5 NXB MOV 8 N7:0 NXB XIO B3:0/5 XIO T4:2/TT BST MOV N9:16 N7:2 NXB RES T4:2 NXB OTL B3:0/5 BND NXB XIC T4:2/DN MOV 35 N7:1 BND EOR
%   N7:1  SEQ_STEP_NUM  "Sequence Step Number" %
%   B3:0/5  ENABLE_SEQ_STEP_TMR  "Enable Sequence Step Timer" %
%   N7:0  SEQ_STEP_OUTPUTS  "Sequence Step Outputs" %
%   T4:2  SEQ_STEP_TIMER  "Sequence Step Timer" %
%   N7:2  SEQ_STEP_TIMER_PRE  "Sequence Step Timer Preset" %

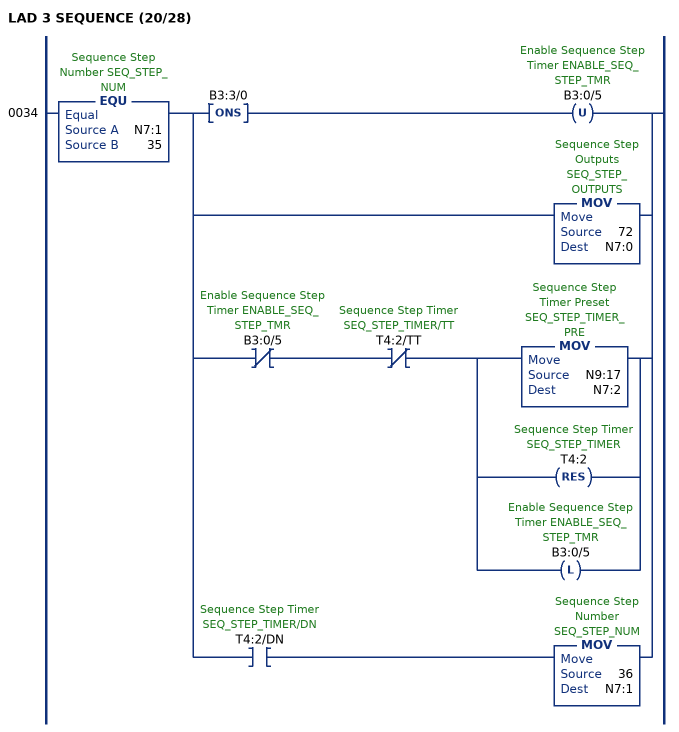
% Rung: 34 %
SOR EQU N7:1 35 BST ONS B3:3/0 OTU B3:0/5 NXB MOV 72 N7:0 NXB XIO B3:0/5 XIO T4:2/TT BST MOV N9:17 N7:2 NXB RES T4:2 NXB OTL B3:0/5 BND NXB XIC T4:2/DN MOV 36 N7:1 BND EOR
%   N7:1  SEQ_STEP_NUM  "Sequence Step Number" %
%   B3:0/5  ENABLE_SEQ_STEP_TMR  "Enable Sequence Step Timer" %
%   N7:0  SEQ_STEP_OUTPUTS  "Sequence Step Outputs" %
%   T4:2  SEQ_STEP_TIMER  "Sequence Step Timer" %
%   N7:2  SEQ_STEP_TIMER_PRE  "Sequence Step Timer Preset" %

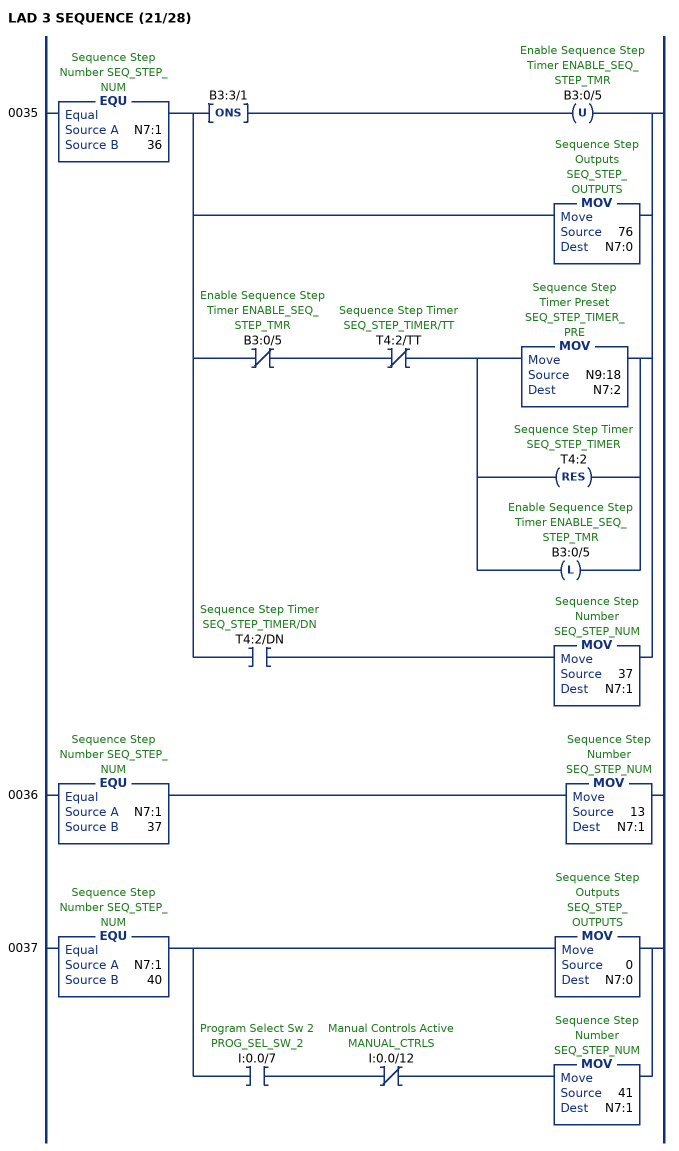
% Rung: 35 %
SOR EQU N7:1 36 BST ONS B3:3/1 OTU B3:0/5 NXB MOV 76 N7:0 NXB XIO B3:0/5 XIO T4:2/TT BST MOV N9:18 N7:2 NXB RES T4:2 NXB OTL B3:0/5 BND NXB XIC T4:2/DN MOV 37 N7:1 BND EOR
%   N7:1  SEQ_STEP_NUM  "Sequence Step Number" %
%   B3:0/5  ENABLE_SEQ_STEP_TMR  "Enable Sequence Step Timer" %
%   N7:0  SEQ_STEP_OUTPUTS  "Sequence Step Outputs" %
%   T4:2  SEQ_STEP_TIMER  "Sequence Step Timer" %
%   N7:2  SEQ_STEP_TIMER_PRE  "Sequence Step Timer Preset" %
% Rung: 36 %
SOR EQU N7:1 37 MOV 13 N7:1 EOR
%   N7:1  SEQ_STEP_NUM  "Sequence Step Number" %
% Rung: 37 %
SOR EQU N7:1 40 BST MOV 0 N7:0 NXB XIC I:0.0/7 XIO I:0.0/12 MOV 41 N7:1 BND EOR
%   N7:1  SEQ_STEP_NUM  "Sequence Step Number" %
%   N7:0  SEQ_STEP_OUTPUTS  "Sequence Step Outputs" %
%   I:0.0/7  PROG_SEL_SW_2  "Program Select Sw 2" %
%   I:0.0/12  MANUAL_CTRLS  "Manual Controls Active" %

